(* IEC 61131-3 sources: test/, 2 files *)

(* ---- FX5U_Motor_Control.st ---- *)
(*
================================================================================
FX5U PLC 电机控制程序 (ST语言)
功能: 电机启动/停止控制，带保护功能和状态指示
作者: PLC程序
日期: 2026-01-11
版本: V1.0
================================================================================
*)

PROGRAM Motor_Control
VAR
    // 输入信号定义
    Start_Button    : BOOL := FALSE;    // 启动按钮 (X0)
    Stop_Button     : BOOL := FALSE;    // 停止按钮 (X1)
    Emergency_Stop  : BOOL := FALSE;    // 急停按钮 (X2) - 常闭触点
    Overload_Relay  : BOOL := FALSE;    // 过载继电器 (X3) - 常闭触点
    Thermal_Switch  : BOOL := FALSE;    // 热保护开关 (X4) - 常闭触点
    Motor_Feedback  : BOOL := FALSE;    // 电机运行反馈 (X5)

    // 输出信号定义
    Motor_Contactor : BOOL := FALSE;    // 电机接触器 (Y0)
    Run_Indicator   : BOOL := FALSE;    // 运行指示灯 (Y1) - 绿灯
    Fault_Indicator : BOOL := FALSE;    // 故障指示灯 (Y2) - 红灯
    Ready_Indicator : BOOL := FALSE;    // 就绪指示灯 (Y3) - 黄灯

    // 内部变量
    Motor_Run_Command   : BOOL := FALSE;    // 电机运行命令
    Protection_OK       : BOOL := FALSE;    // 保护条件正常
    Start_Condition     : BOOL := FALSE;    // 启动条件
    Stop_Condition      : BOOL := FALSE;    // 停止条件
    Fault_Status        : BOOL := FALSE;    // 故障状态

    // 定时器变量
    Start_Delay_Timer   : TON;              // 启动延时定时器
    Fault_Reset_Timer   : TON;              // 故障复位定时器

    // 定时器时间常数
    START_DELAY_TIME    : TIME := T#500ms;  // 启动延时时间
    FAULT_RESET_TIME    : TIME := T#3s;     // 故障复位时间
END_VAR

BEGIN
    // ========== 保护条件检查 ==========
    // 检查所有保护输入（常闭触点，正常时为TRUE）
    Protection_OK := Emergency_Stop AND Overload_Relay AND Thermal_Switch;

    // ========== 故障检测 ==========
    // 故障条件：任一保护条件不满足
    Fault_Status := NOT Protection_OK;

    // ========== 启动条件判断 ==========
    // 启动条件：按下启动按钮 且 保护正常 且 无故障状态
    Start_Condition := Start_Button AND Protection_OK AND NOT Fault_Status;

    // ========== 停止条件判断 ==========
    // 停止条件：按下停止按钮 或 出现故障
    Stop_Condition := Stop_Button OR Fault_Status;

    // ========== 电机控制逻辑 ==========
    // 启动延时定时器
    Start_Delay_Timer(
        IN := Start_Condition AND NOT Motor_Run_Command,
        PT := START_DELAY_TIME
    );

    // 电机运行命令 - 自保持逻辑
    IF Start_Delay_Timer.Q THEN
        Motor_Run_Command := TRUE;
    ELSIF Stop_Condition THEN
        Motor_Run_Command := FALSE;
    END_IF;

    // 电机接触器输出
    Motor_Contactor := Motor_Run_Command AND Protection_OK;

    // ========== 故障复位逻辑 ==========
    // 故障复位定时器 - 故障消除后自动复位
    Fault_Reset_Timer(
        IN := Protection_OK AND Fault_Status,
        PT := FAULT_RESET_TIME
    );

    // 故障状态复位
    IF Fault_Reset_Timer.Q THEN
        Fault_Status := FALSE;
    END_IF;

    // ========== 状态指示灯控制 ==========

    // 就绪指示灯（黄灯）- 系统正常但电机未运行
    Ready_Indicator := Protection_OK AND NOT Motor_Run_Command AND NOT Fault_Status;

    // 运行指示灯（绿灯）- 电机正在运行
    Run_Indicator := Motor_Contactor AND Motor_Feedback;

    // 故障指示灯（红灯）- 系统故障
    Fault_Indicator := Fault_Status;

END_PROGRAM

(*
================================================================================
I/O 分配表:
================================================================================
输入 (X):
X0 - Start_Button      启动按钮 (常开)
X1 - Stop_Button       停止按钮 (常开)
X2 - Emergency_Stop    急停按钮 (常闭)
X3 - Overload_Relay    过载继电器 (常闭)
X4 - Thermal_Switch    热保护开关 (常闭)
X5 - Motor_Feedback    电机运行反馈 (常开)

输出 (Y):
Y0 - Motor_Contactor   电机接触器
Y1 - Run_Indicator     运行指示灯 (绿灯)
Y2 - Fault_Indicator   故障指示灯 (红灯)
Y3 - Ready_Indicator   就绪指示灯 (黄灯)

================================================================================
功能说明:
================================================================================
1. 启动功能:
   - 按下启动按钮，系统检查保护条件
   - 保护正常时，延时500ms后启动电机
   - 电机启动后自保持运行

2. 停止功能:
   - 按下停止按钮立即停止电机
   - 任何保护条件触发时自动停止

3. 保护功能:
   - 急停保护：急停按钮按下时立即停止
   - 过载保护：过载继电器动作时停止电机
   - 热保护：热保护开关动作时停止电机
   - 故障自动复位：故障消除3秒后自动复位

4. 状态指示:
   - 黄灯：系统就绪，可以启动
   - 绿灯：电机正常运行
   - 红灯：系统故障

================================================================================
使用说明:
================================================================================
1. 将此程序下载到FX5U PLC中
2. 按照I/O分配表连接外部设备
3. 确保所有保护设备正常连接
4. 上电后观察指示灯状态
5. 按启动按钮启动电机，按停止按钮停止电机

注意事项:
- 急停、过载、热保护均为常闭触点
- 电机反馈信号用于确认电机实际运行状态
- 故障时红灯亮，故障消除后会自动复位
================================================================================
*)

(* ---- PLC_Program_Template.st ---- *)
(*
================================================================================
PLC程序开发模板 - ST语言
================================================================================
项目名称: [在此填写项目名称]
功能描述: [在此描述程序功能]
作者: [作者名称]
创建日期: [YYYY-MM-DD]
版本: V1.0
最后修改: [YYYY-MM-DD]
================================================================================
修改记录:
V1.0 - [日期] - [作者] - 初始版本
================================================================================
*)

PROGRAM [程序名称]
VAR
    //==========================================================================
    // 输入信号定义 (Input Signals)
    //==========================================================================
    // 按钮输入 (Push Buttons)
    gStart_Button       : BOOL := FALSE;    // 启动按钮 (X0)
    gStop_Button        : BOOL := FALSE;    // 停止按钮 (X1)
    gReset_Button       : BOOL := FALSE;    // 复位按钮 (X2)

    // 保护输入 (Protection Inputs) - 常闭触点
    gEmergency_Stop     : BOOL := FALSE;    // 急停按钮 (X3) - NC
    gOverload_Relay     : BOOL := FALSE;    // 过载继电器 (X4) - NC
    gThermal_Switch     : BOOL := FALSE;    // 热保护开关 (X5) - NC

    // 反馈输入 (Feedback Inputs)
    gDevice_Feedback    : BOOL := FALSE;    // 设备运行反馈 (X6)
    gPosition_Sensor    : BOOL := FALSE;    // 位置传感器 (X7)

    // 模拟量输入 (Analog Inputs)
    gAnalog_Input_1     : INT := 0;         // 模拟量输入1 (AD0)
    gAnalog_Input_2     : INT := 0;         // 模拟量输入2 (AD1)

    //==========================================================================
    // 输出信号定义 (Output Signals)
    //==========================================================================
    // 控制输出 (Control Outputs)
    gMain_Contactor     : BOOL := FALSE;    // 主接触器 (Y0)
    gAux_Contactor      : BOOL := FALSE;    // 辅助接触器 (Y1)
    gValve_Output       : BOOL := FALSE;    // 阀门输出 (Y2)

    // 指示灯输出 (Indicator Outputs)
    gRun_Indicator      : BOOL := FALSE;    // 运行指示灯 (Y3) - 绿灯
    gFault_Indicator    : BOOL := FALSE;    // 故障指示灯 (Y4) - 红灯
    gReady_Indicator    : BOOL := FALSE;    // 就绪指示灯 (Y5) - 黄灯

    // 报警输出 (Alarm Outputs)
    gAlarm_Horn         : BOOL := FALSE;    // 报警蜂鸣器 (Y6)
    gAlarm_Light        : BOOL := FALSE;    // 报警灯 (Y7)

    // 模拟量输出 (Analog Outputs)
    gAnalog_Output_1    : INT := 0;         // 模拟量输出1 (DA0)
    gAnalog_Output_2    : INT := 0;         // 模拟量输出2 (DA1)

    //==========================================================================
    // 内部变量定义 (Internal Variables)
    //==========================================================================
    // 控制逻辑变量 (Control Logic Variables)
    System_Enable       : BOOL := FALSE;    // 系统使能
    Run_Command         : BOOL := FALSE;    // 运行命令
    Protection_OK       : BOOL := FALSE;    // 保护条件正常
    Start_Condition     : BOOL := FALSE;    // 启动条件
    Stop_Condition      : BOOL := FALSE;    // 停止条件

    // 状态变量 (Status Variables)
    System_State        : INT := 0;         // 系统状态 (0:停止, 1:启动中, 2:运行, 99:故障)
    Fault_Code          : INT := 0;         // 故障代码
    Operation_Mode      : INT := 1;         // 操作模式 (1:手动, 2:自动)

    // 故障检测变量 (Fault Detection Variables)
    Fault_Status        : BOOL := FALSE;    // 故障状态
    Emergency_Fault     : BOOL := FALSE;    // 急停故障
    Overload_Fault      : BOOL := FALSE;    // 过载故障
    Thermal_Fault       : BOOL := FALSE;    // 热保护故障
    Timeout_Fault       : BOOL := FALSE;    // 超时故障

    //==========================================================================
    // 定时器定义 (Timer Definitions)
    //==========================================================================
    Start_Delay_Timer   : TON;              // 启动延时定时器
    Stop_Delay_Timer    : TON;              // 停止延时定时器
    Fault_Reset_Timer   : TON;              // 故障复位定时器
    Watchdog_Timer      : TON;              // 看门狗定时器
    Blink_Timer         : TON;              // 闪烁定时器

    //==========================================================================
    // 计数器定义 (Counter Definitions)
    //==========================================================================
    Start_Counter       : CTU;              // 启动次数计数器
    Fault_Counter       : CTU;              // 故障次数计数器

    //==========================================================================
    // 时间常数定义 (Time Constants)
    //==========================================================================
    START_DELAY_TIME    : TIME := T#500ms;  // 启动延时时间
    STOP_DELAY_TIME     : TIME := T#200ms;  // 停止延时时间
    FAULT_RESET_TIME    : TIME := T#3s;     // 故障复位时间
    WATCHDOG_TIME       : TIME := T#5s;     // 看门狗时间
    BLINK_TIME          : TIME := T#500ms;  // 闪烁周期

    //==========================================================================
    // 数值常数定义 (Numeric Constants)
    //==========================================================================
    MAX_START_COUNT     : INT := 100;       // 最大启动次数
    MAX_FAULT_COUNT     : INT := 10;        // 最大故障次数
    ANALOG_MIN_VALUE    : INT := 0;         // 模拟量最小值
    ANALOG_MAX_VALUE    : INT := 4000;      // 模拟量最大值

END_VAR

BEGIN
    //==========================================================================
    // 程序主体 (Main Program Body)
    //==========================================================================

    (* ========== 系统初始化 ========== *)
    // 在此添加系统初始化代码

    (* ========== 输入信号处理 ========== *)
    // 在此添加输入信号滤波、边沿检测等处理

    (* ========== 保护条件检查 ========== *)
    // 检查所有保护输入（常闭触点，正常时为TRUE）
    Protection_OK := gEmergency_Stop AND gOverload_Relay AND gThermal_Switch;

    // 故障检测
    Emergency_Fault := NOT gEmergency_Stop;
    Overload_Fault := NOT gOverload_Relay;
    Thermal_Fault := NOT gThermal_Switch;

    // 综合故障状态
    Fault_Status := Emergency_Fault OR Overload_Fault OR Thermal_Fault OR Timeout_Fault;

    (* ========== 启动/停止条件判断 ========== *)
    // 启动条件：按下启动按钮 且 保护正常 且 无故障状态 且 系统使能
    Start_Condition := gStart_Button AND Protection_OK AND NOT Fault_Status AND System_Enable;

    // 停止条件：按下停止按钮 或 出现故障
    Stop_Condition := gStop_Button OR Fault_Status;

    (* ========== 主控制逻辑 ========== *)
    // 在此添加主要的控制逻辑

    (* ========== 定时器处理 ========== *)
    // 启动延时定时器
    Start_Delay_Timer(
        IN := Start_Condition AND NOT Run_Command,
        PT := START_DELAY_TIME
    );

    // 故障复位定时器
    Fault_Reset_Timer(
        IN := Protection_OK AND Fault_Status,
        PT := FAULT_RESET_TIME
    );

    // 闪烁定时器
    Blink_Timer(
        IN := TRUE,
        PT := BLINK_TIME
    );

    (* ========== 计数器处理 ========== *)
    // 启动次数计数
    Start_Counter(
        CU := Start_Delay_Timer.Q,
        RESET := gReset_Button,
        PV := MAX_START_COUNT
    );

    (* ========== 状态机控制 ========== *)
    CASE System_State OF
        0: // 停止状态
            IF Start_Delay_Timer.Q THEN
                System_State := 1;
            END_IF;

        1: // 启动中状态
            // 在此添加启动序列逻辑
            System_State := 2; // 直接进入运行状态（示例）

        2: // 运行状态
            IF Stop_Condition THEN
                System_State := 0;
            END_IF;

        99: // 故障状态
            IF Fault_Reset_Timer.Q THEN
                System_State := 0;
            END_IF;

        ELSE
            System_State := 0; // 默认返回停止状态
    END_CASE;

    (* ========== 输出控制 ========== *)
    // 主要输出控制
    gMain_Contactor := (System_State = 2) AND Protection_OK;

    // 指示灯控制
    gReady_Indicator := (System_State = 0) AND Protection_OK AND NOT Fault_Status;
    gRun_Indicator := (System_State = 2);
    gFault_Indicator := Fault_Status OR (System_State = 99);

    // 报警输出控制
    gAlarm_Horn := Fault_Status AND Blink_Timer.Q;
    gAlarm_Light := Fault_Status;

    (* ========== 模拟量处理 ========== *)
    // 在此添加模拟量输入处理和输出控制

    (* ========== 通信处理 ========== *)
    // 在此添加通信相关代码

    (* ========== 数据记录 ========== *)
    // 在此添加数据记录和历史数据处理

END_PROGRAM

(*
================================================================================
I/O 分配表 (I/O Assignment Table)
================================================================================
输入 (Inputs):
X0  - gStart_Button       启动按钮 (常开)
X1  - gStop_Button        停止按钮 (常开)
X2  - gReset_Button       复位按钮 (常开)
X3  - gEmergency_Stop     急停按钮 (常闭)
X4  - gOverload_Relay     过载继电器 (常闭)
X5  - gThermal_Switch     热保护开关 (常闭)
X6  - gDevice_Feedback    设备运行反馈 (常开)
X7  - gPosition_Sensor    位置传感器 (常开)

输出 (Outputs):
Y0  - gMain_Contactor     主接触器
Y1  - gAux_Contactor      辅助接触器
Y2  - gValve_Output       阀门输出
Y3  - gRun_Indicator      运行指示灯 (绿灯)
Y4  - gFault_Indicator    故障指示灯 (红灯)
Y5  - gReady_Indicator    就绪指示灯 (黄灯)
Y6  - gAlarm_Horn         报警蜂鸣器
Y7  - gAlarm_Light        报警灯

模拟量 (Analog):
AD0 - gAnalog_Input_1     模拟量输入1
AD1 - gAnalog_Input_2     模拟量输入2
DA0 - gAnalog_Output_1    模拟量输出1
DA1 - gAnalog_Output_2    模拟量输出2

================================================================================
使用说明 (Usage Instructions)
================================================================================
1. 复制此模板文件并重命名为具体项目名称
2. 修改头部注释中的项目信息
3. 根据实际需求修改变量定义和I/O分配
4. 在对应的程序段中添加具体的控制逻辑
5. 更新I/O分配表以匹配实际硬件连接
6. 测试程序并记录修改历史

注意事项 (Notes):
- 保护输入均为常闭触点，正常时为TRUE
- 所有定时器和计数器都有对应的复位条件
- 状态机设计便于扩展和维护
- 变量命名遵循统一的命名规范
- 包含完整的故障检测和处理机制
================================================================================
*)
